Yaskawa INFORM job: R1_W27-A4(90,180)_KM_OKR2.JBI

/JOB
//NAME R1_W27-A4(90,180)_KM_OKR2
///FOLDERNAME KRIS-SCIANA
//POS
///NPOS 128,128,0,5,0,0
///TOOL 0
///POSTYPE PULSE
///PULSE
C00000=44200,21638,-8218,30156,108783,8626
C00001=67595,-7097,-4564,35957,72928,-14479
C00002=80598,-11631,1969,12944,68774,-20478
C00003=71791,13613,26980,27330,77562,-23201
C00004=71369,36291,48447,29991,82050,-38866
C00005=71229,45479,49804,30590,69224,-77746
C00006=71229,48407,56883,31154,66760,-78457
C00007=70619,60634,70702,31805,69801,-77954
C00008=71209,58588,68328,31698,69934,-77673
C00009=70997,59310,69162,31736,69890,-77772
C00010=70997,61787,74250,32090,68300,-78245
C00011=70997,57612,65507,31493,71070,-77426
C00012=71229,45479,49804,30590,69224,-77746
C00013=71791,13613,26980,27330,77562,-23201
C00014=80598,-11631,1969,12944,68774,-20478
C00015=80599,-10712,4409,13031,67770,-20590
C00016=81000,-9857,5799,13000,67300,-20494
C00017=81299,-8771,6650,12945,67285,-20385
C00018=81000,-9857,5799,13000,67300,-20494
C00019=81000,-9326,7151,13051,66755,-20556
C00020=81000,-9857,5799,13000,67300,-20494
C00021=75972,1459,14259,17611,75755,-34351
C00022=77593,2438,17479,17632,73999,-34024
C00023=78143,1669,16828,17600,73886,-33841
C00024=76339,1181,13702,17577,75868,-34199
C00025=80626,-10617,4483,1955,54639,1218
C00026=80604,-16221,-12250,12512,75016,-19809
C00027=77456,-21668,-17293,6564,52888,-78355
C00028=80617,-10651,4457,5429,44969,-77444
C00029=80614,-10662,4448,5430,44969,-77445
C00030=78880,-15057,3874,9656,39826,-78954
C00031=81168,-10487,5664,5147,44277,-77224
C00032=80549,-11563,2448,5400,45738,-77430
C00033=80742,-8639,8257,8065,40593,-77243
C00034=80443,-9972,5851,8148,41408,-77313
C00035=78226,-16015,-2651,9320,43747,-78172
C00036=65744,24754,34700,31474,70065,-79759
C00037=68185,33051,42925,31367,68479,-79216
C00038=70799,57683,71232,35631,65009,-79625
C00039=70611,44259,48623,30654,69536,-77912
C00040=75134,-17482,-5239,8428,47880,-79749
C00041=60313,-1918,20521,42182,54711,-86083
C00042=62757,5453,32917,43679,50705,-86826
C00043=62432,2076,32536,48578,48674,-88823
C00044=72918,-15655,19579,49112,42093,-86873
C00045=73223,-16448,18995,49076,41906,-86801
C00046=67737,-13796,25454,59346,48360,-88683
C00047=63268,-14792,20282,57576,52355,-88326
C00048=77858,-26804,-24776,6192,54811,-78068
C00049=77858,-26804,-24776,6192,54811,8206
C00050=80560,-10852,4301,23089,88681,-39643
C00051=80562,-10848,4304,23089,88680,-39643
C00052=78564,-17199,-442,25373,86442,-37023
C00053=80047,-12757,2574,23029,88900,-39787
C00054=79798,-9411,5485,22999,88903,-39877
C00055=73541,-21178,5085,31179,78420,-45097
C00056=72021,-21514,1829,31651,80058,-45695
C00057=88031,-24585,-19769,24865,79157,-46389
C00058=74088,-80099,-54440,46439,68409,-50026
C00059=71054,-82284,-78741,37326,78086,-53143
C00060=71054,-82284,-78741,37326,78086,-53143
C00061=141655,19461,21674,-54626,60929,-83209
C00062=140768,21158,24027,-54713,60067,-83168
C00063=140768,21810,26002,-55124,59545,-82791
C00064=140768,21158,24027,-54713,60067,-83168
C00065=155664,19148,-9811,-52803,80751,-87559
C00066=155140,18500,-10419,-52658,80490,-87680
C00067=155664,19148,-9811,-52803,80751,-87559
C00068=158287,-4573,8654,-106143,62454,-35624
C00069=144891,16645,-13127,-43951,85052,9819
C00070=144769,17601,-12243,-43922,84955,9807
C00071=144891,16645,-13127,-43951,85052,9819
C00072=120685,-15723,-29307,-37667,68905,5594
C00073=124617,-55133,-52955,-40369,66182,8461
C00074=97830,-52515,-57171,7086,69913,-23311
C00075=85987,-45740,-53193,41668,69314,-45492
C00076=79888,-2056,-15574,47948,58225,-80763
C00077=84628,7663,-5674,40179,60293,-77610
C00078=84628,7673,-5553,40205,60240,-77633
C00079=84628,7816,-4041,40518,59580,-77920
C00080=84628,7673,-5553,40205,60240,-77633
C00081=85256,7940,-5318,39944,59945,-77448
C00082=84628,7673,-5553,40205,60240,-77633
C00083=84548,-2926,-17409,39122,61468,-76703
C00084=90189,-10947,-19792,34314,54151,-73686
C00085=87731,11667,-738,31608,52128,-71965
C00086=84586,20469,7503,37448,56009,-75800
C00087=80660,6659,-12646,40128,64767,-77184
C00088=80660,6659,-12646,40128,64767,11736
C00089=73617,-18493,-32865,42959,67690,9655
C00090=69872,-47770,-49426,45593,66014,7010
C00091=99316,-51214,-54357,3838,55594,8091
C00092=108651,-54494,-53004,-14245,50847,11455
C00093=128597,-2596,-22816,-39758,74552,6944
C00094=106236,1119,-8655,-33108,59628,2381
C00095=100502,1007,-8349,-30553,57262,531
C00096=121335,-11193,4016,-73235,33107,-65970
C00097=121314,-11175,4070,-52209,41640,-77705
C00098=121322,-11192,4065,-52217,41640,-77699
C00099=121326,-11199,4064,-52221,41641,-77697
C00100=121319,-11903,2209,-51536,42130,-78112
C00101=122361,-11180,4070,-52628,42228,-77380
C00102=121327,-11199,4064,-52222,41641,-77696
C00103=121327,-11199,4064,-52222,41641,-77696
C00104=121328,-11199,4065,-52223,41641,-77696
C00105=121325,-11192,4067,-52219,41641,-77698
C00106=121317,-11174,4072,-52211,41640,-77704
C00107=121324,-11180,4031,-66023,34984,-69858
C00108=121305,-11164,4064,-33775,34107,58027
C00109=121211,-10931,3851,-41868,44478,53115
C00110=117301,-6994,3549,-31202,46743,49457
C00111=116677,-5672,6257,-33160,45686,49655
C00112=121892,-11860,2463,-42413,44821,53021
C00113=122357,-11331,3957,-43061,44562,53464
C00114=117167,2531,12951,-33359,45962,49818
C00115=117195,3946,14157,-33381,45960,49835
C00116=119475,-2324,8124,-34252,47278,50538
C00117=123076,-13488,2301,-43433,44847,53751
C00118=121299,-11171,4074,-39219,33281,58177
C00119=116680,2407,14742,-33067,37032,-10813
C00120=123012,16327,32624,-57039,46741,-7607
C00121=119054,23161,42484,-58310,42982,-7235
C00122=115883,23536,42847,-57561,41091,-8058
C00123=120097,16950,35052,-57333,44360,-7727
C00124=131063,-12359,7007,-57867,52103,-6183
C00125=129161,-93141,-40285,-63646,27916,71647
C00126=59909,-160831,-87956,-63646,27916,71647
C00127=39710,-191418,-114720,-5142,50077,71647
BC00000=114828,529484,1075169
BC00001=111963,471444,1075173
BC00002=110304,437827,1075175
BC00003=110304,437827,1075175
BC00004=110304,437827,1075175
BC00005=81757,444144,1016188
BC00006=81757,444144,1016188
BC00007=81757,444144,1016188
BC00008=81757,444144,1016188
BC00009=81757,444144,1016188
BC00010=81757,444144,1016188
BC00011=81757,444144,1016188
BC00012=81757,444144,1016188
BC00013=110304,437827,1075175
BC00014=110304,437827,1075175
BC00015=109200,433065,1065059
BC00016=108759,431160,1056755
BC00017=108759,431160,1056755
BC00018=108759,431160,1056755
BC00019=108759,431160,1056755
BC00020=108759,431160,1056755
BC00021=119290,430574,1053953
BC00022=119290,430574,1053953
BC00023=119290,430574,1053953
BC00024=119290,430574,1053953
BC00025=69199,447701,1057682
BC00026=110304,437827,1075175
BC00027=82308,447284,1075175
BC00028=81837,447193,1052280
BC00029=81780,445015,1026500
BC00030=81757,444144,1016188
BC00031=81757,444144,1016188
BC00032=81757,444144,1016188
BC00033=81757,444144,1016188
BC00034=81757,444144,1016188
BC00035=81757,444144,1016188
BC00036=81757,444144,1016188
BC00037=81757,444144,1016188
BC00038=81757,444144,1016188
BC00039=81757,444144,1016188
BC00040=82300,439412,1075174
BC00041=82300,439412,1075174
BC00042=82300,439412,1075174
BC00043=82300,439412,1075174
BC00044=82300,439412,1075174
BC00045=82300,439412,1075174
BC00046=82300,439412,1075174
BC00047=82300,439412,1075174
BC00048=82308,447284,1075175
BC00049=82308,447284,1075175
BC00050=162842,405450,1047947
BC00051=157631,403387,1028943
BC00052=155626,402592,1021627
BC00053=155546,402561,1021342
BC00054=155546,402561,1021342
BC00055=155554,402564,1021370
BC00056=155546,402561,1021342
BC00057=169608,431160,979206
BC00058=162842,405450,1047947
BC00059=169608,545788,979206
BC00060=169608,545788,42321
BC00061=261853,469584,216144
BC00062=261853,469584,216144
BC00063=261853,469584,216144
BC00064=261853,469584,216144
BC00065=307725,459293,22582
BC00066=307725,459293,22582
BC00067=307725,459293,22582
BC00068=299050,464357,35683
BC00069=289567,469892,50003
BC00070=289567,469892,50003
BC00071=289567,469892,50003
BC00072=193210,455841,135951
BC00073=193210,455841,135951
BC00074=193210,455841,135951
BC00075=193210,455841,135951
BC00076=141494,455846,135950
BC00077=141494,455846,135950
BC00078=141494,455846,135950
BC00079=141494,455846,135950
BC00080=141494,455846,135950
BC00081=141494,455846,135950
BC00082=141494,455846,135950
BC00083=141978,455876,135765
BC00084=141978,455876,135765
BC00085=141978,455876,135765
BC00086=141978,455876,135765
BC00087=141978,455876,135765
BC00088=141978,455876,135765
BC00089=141978,455876,135765
BC00090=141978,455876,135765
BC00091=184986,458555,119298
BC00092=184986,458555,119298
BC00093=232126,461491,101248
BC00094=174559,453133,152583
BC00095=158444,451963,159769
BC00096=191752,502679,198110
BC00097=212977,452054,280459
BC00098=218243,449415,262530
BC00099=220349,448360,255359
BC00100=220349,448360,255359
BC00101=220349,448360,255359
BC00102=220340,443751,255365
BC00103=220339,443318,255365
BC00104=220329,438710,255371
BC00105=218223,439765,262543
BC00106=212957,442404,280472
BC00107=194357,497799,228108
BC00108=206310,480373,286705
BC00109=214934,438060,283714
BC00110=214934,438060,283714
BC00111=214934,438060,283714
BC00112=221705,433918,270833
BC00113=221705,433918,270833
BC00114=214934,438060,283714
BC00115=214934,438060,283714
BC00116=214934,438060,283714
BC00117=212593,431556,287024
BC00118=215962,481703,300457
BC00119=215962,481703,300457
BC00120=215962,481703,300457
BC00121=215962,481703,300457
BC00122=215962,481703,300457
BC00123=215962,481703,300457
BC00124=215962,481703,300457
BC00125=215962,481703,300457
BC00126=215962,481703,300457
BC00127=225321,555844,754221
///POSTYPE BASE
///RECTAN
///RCONF 0,0,0,0,1,0,0,0,0,0,0,0,0,0,0,0,0,0,0,0,0,0,0,0
P00006=2.006,1.622,-0.565,0.0000,0.0000,0.0000
///RCONF 0,0,0,0,0,0,0,0,0,0,0,0,0,0,0,0,0,0,0,0,0,0,0,0
P00014=4.542,-3.738,3.339,0.0000,0.0000,0.0000
P00015=5.923,-0.025,-0.886,0.0000,0.0000,0.0000
///RCONF 0,0,0,0,1,0,0,0,0,0,0,0,0,0,0,0,0,0,0,0,0,0,0,0
P00021=0.073,2.058,-0.109,0.0000,0.0000,0.0000
///RCONF 0,0,0,0,0,0,0,0,0,0,0,0,0,0,0,0,0,0,0,0,0,0,0,0
P00030=-0.014,-0.768,0.131,0.0000,0.0000,0.0000
//INST
///DATE 2025/04/17 14:03
///ATTR SC,RW
///GROUP1 RB1,BS1
NOP
'r2_W27-A4(90,180)
'
'Path S896
SFTOF
MOVJ C00000 BC00000 VJ=50.00
MOVJ C00001 BC00001 VJ=50.00
MOVL C00002 BC00002 V=100.0
MOVL C00003 BC00003 V=100.0
MOVL C00004 BC00004 V=100.0
MOVL C00005 BC00005 V=100.0
MOVL C00006 BC00006 V=100.0
MOVL C00007 BC00007 V=100.0
REFP 3 C00008 BC00008
CALL JOB:SEARCH-R1
SET P015 P006
SFTON P015
MOVL C00009 BC00009 V=100.0
REFP 3 C00010 BC00010
CALL JOB:SEARCH-R1
SET P015 P006
SFTON P015
MOVL C00011 BC00011 V=100.0
MOVL C00012 BC00012 V=100.0
MOVL C00013 BC00013 V=100.0
MOVL C00014 BC00014 V=100.0
MOVL C00015 BC00015 V=100.0
MOVL C00016 BC00016 V=60.0
REFP 3 C00017 BC00017
CALL JOB:SEARCH-R1
SET P014 P006
SFTON P014
MOVL C00018 BC00018 V=100.0
REFP 3 C00019 BC00019
CALL JOB:SEARCH-R1
SET P014 P006
SFTON P014
MOVL C00020 BC00020 V=100.0
MOVL C00021 BC00021 V=100.0
MOVL C00022 BC00022 V=100.0
REFP 3 C00023 BC00023
CALL JOB:SEARCH-R1
SET P014 P006
SFTON P014
MOVL C00024 BC00024 V=100.0
MOVL C00025 BC00025 V=100.0
'Path VIA902
SFTOF
MOVJ C00026 BC00026 VJ=20.00
'Path W898
SFTOF
SFTON P014
MOVJ C00027 BC00027 VJ=20.00
MOVJ C00028 BC00028 VJ=20.00
MOVL C00029 BC00029 V=100.0
MOVL C00030 BC00030 V=166.7 PL=0
REFP 1 C00031 BC00031
REFP 2 C00032 BC00032
MACRO1 MJ#(0) ARGF7
COMM ARCON
MOVL C00033 BC00033 V=10.0
ARCOF
MOVL C00034 BC00034 V=166.7
MOVL C00035 BC00035 V=166.7
SFTON P014
MOVL C00036 BC00036 V=83.3
ARCON
MOVL C00037 BC00037 V=9.2
SFTON P015
MOVL C00038 BC00038 V=9.2
ARCOF
MOVL C00039 BC00039 V=200.0
MOVL C00040 BC00040 V=400.0
SFTOF
MOVJ C00041 BC00041 VJ=20.00
SFTON P014
MOVJ C00042 BC00042 VJ=10.00
ARCON
MOVL C00043 BC00043 V=9.2
MOVL C00044 BC00044 V=9.2
MOVL C00045 BC00045 V=9.2
MOVL C00046 BC00046 V=9.2
ARCOF
MOVJ C00047 BC00047 VJ=10.00
'Path VIA903
SFTOF
MOVJ C00048 BC00048 VJ=20.00
'Path VIA904
SFTOF
MOVJ C00049 BC00049 VJ=20.00
'Path W901
SFTOF
SFTON P014
MOVJ C00050 BC00050 VJ=20.00
MOVL C00051 BC00051 V=100.0
MOVL C00052 BC00052 V=100.0 PL=0
REFP 1 C00053 BC00053
REFP 2 C00054 BC00054
MACRO1 MJ#(0) ARGF6
COMM ARCON
MOVL C00055 BC00055 V=11.7
ARCOF
MOVL C00056 BC00056 V=100.0
MOVL C00057 BC00057 V=100.0
SFTOF
'Path VIA907
SFTOF
MOVJ C00058 BC00058 VJ=20.00
'Path VIA905
SFTOF
MOVJ C00059 BC00059 VJ=100.00
CALL JOB:CLEAN-R1_LONG
'Path VIA906
SFTOF
MOVJ C00060 BC00060 VJ=100.00
'Path S845
SFTOF
MOVL C00061 BC00061 V=133.3
MOVL C00062 BC00062 V=60.0
REFP 3 C00063 BC00063
CALL JOB:SEARCH-R1
SET P021 P006
SFTON P021
MOVL C00064 BC00064 V=60.0
MOVL C00065 BC00065 V=100.0
REFP 3 C00066 BC00066
CALL JOB:SEARCH-R1
SET P021 P006
SFTON P021
MOVL C00067 BC00067 V=100.0
MOVL C00068 BC00068 V=100.0
MOVL C00069 BC00069 V=100.0
REFP 3 C00070 BC00070
CALL JOB:SEARCH-R1
SET P021 P006
SFTON P021
MOVL C00071 BC00071 V=60.0
SFTOF
MOVJ C00072 BC00072 VJ=10.00
MOVJ C00073 BC00073 VJ=10.00
MOVJ C00074 BC00074 VJ=10.00
MOVJ C00075 BC00075 VJ=10.00
MOVJ C00076 BC00076 VJ=10.00
MOVJ C00077 BC00077 VJ=10.00
'POMIAR
MOVL C00078 BC00078 V=83.3
REFP 3 C00079 BC00079
CALL JOB:SEARCH-R1
SET P030 P006
SFTON P030
MOVL C00080 BC00080 V=83.3
REFP 3 C00081 BC00081
CALL JOB:SEARCH-R1
SET P030 P006
SFTON P030
MOVL C00082 BC00082 V=83.3
SFTOF
SFTON P030
MOVJ C00083 BC00083 VJ=10.00
MACRO1 MJ#(0) ARGF7
MOVJ C00084 BC00084 VJ=10.00
ARCON
MOVL C00085 BC00085 V=7.5
MOVL C00086 BC00086 V=7.5
ARCOF
MOVJ C00087 BC00087 VJ=10.00
SFTOF
MOVJ C00088 BC00088 VJ=20.00
MOVJ C00089 BC00089 VJ=20.00
MOVJ C00090 BC00090 VJ=20.00
MOVJ C00091 BC00091 VJ=30.00
MOVJ C00092 BC00092 VJ=30.00
MOVL C00093 BC00093 V=100.0
MOVL C00094 BC00094 V=100.0
MOVL C00095 BC00095 V=100.0
'Path W846
SFTOF
SFTON P021
MOVJ C00096 BC00096 VJ=20.00
MOVL C00097 BC00097 V=100.0
MOVL C00098 BC00098 V=100.0
MOVL C00099 BC00099 V=100.0 PL=0
REFP 1 C00100 BC00100
REFP 2 C00101 BC00101
MACRO1 MJ#(0) ARGF0
COMM ARCON
MOVL C00102 BC00102 V=10.0
MOVL C00103 BC00103 V=10.0
MOVL C00104 BC00104 V=10.0
ARCOF
MOVL C00105 BC00105 V=100.0
MOVL C00106 BC00106 V=100.0
MOVL C00107 BC00107 V=100.0
SFTOF
'Path W847
SFTOF
SFTON P021
MOVJ C00108 BC00108 VJ=20.00
MOVL C00109 BC00109 V=100.0
MOVL C00110 BC00110 V=100.0
MOVL C00111 BC00111 V=100.0 PL=0
REFP 1 C00112 BC00112
REFP 2 C00113 BC00113
MACRO1 MJ#(0) ARGF7
COMM ARCON
MOVL C00114 BC00114 V=8.3
MOVL C00115 BC00115 V=8.3
ARCOF
SFTOF
MOVL C00116 BC00116 V=100.0
MOVL C00117 BC00117 V=100.0
MOVJ C00118 BC00118 VJ=20.00
MOVJ C00119 BC00119 VJ=30.00
MOVJ C00120 BC00120 VJ=20.00
MACRO1 MJ#(0) ARGF7
MOVJ C00121 BC00121 VJ=10.00
COMM ARCON
MOVL C00122 BC00122 V=8.3
ARCOF
MOVJ C00123 BC00123 VJ=10.00
SFTOF
MOVJ C00124 BC00124 VJ=40.00
MOVJ C00125 BC00125 VJ=40.00
MOVJ C00126 BC00126 VJ=100.00
MOVJ C00127 BC00127 VJ=100.00
END
